// TIA Portal V20 export
DATA_BLOCK "ControlNodes"   // DB77
{ DB_Accessible_From_OPC_UA := 'FALSE' }
AUTHOR : ERsystem_FA2_DH. Kim
// stored: DBAccessibleFromOPCUA false, DBAccessibleFromWebserver false, MemoryReserve 100, Namespace Unit1.Em3
   VAR
      em { ExternalWritable := 'False'} : "LAF_typeEmControlNode";
      cm : Struct
         Interlock : Struct
            compensatorAxisX : "LER_typeAxisInterlock";
            masterVirtualAxis : "LER_typeAxisInterlock";
            unwinderVirtualAxis : "LER_typeAxisInterlock";
            dancerFwdBwd : "LER_typeTwoWayActInterlock";
            sepaUnwinderIonizerTop : "LER_typeTwoWayActInterlock";
            sepaUnwinderIonizerBottom : "LER_typeTwoWayActInterlock";
         END_STRUCT;
         command : Struct
            compensatorAxisX : "LER_typeAxisCommand";
            masterVirtualAxis : "LER_typeAxisCommand";
            unwinderVirtualAxis : "LER_typeAxisCommand";
            dancerFwdBwd : "LER_typeTwoWayActCommand";
            sepaUnwinderIonizerTop : "LER_typeTwoWayActCommand";
            sepaUnwinderIonizerBottom : "LER_typeTwoWayActCommand";
         END_STRUCT;
         softCam : "Unit1.type_emRelations_em3_SoftCam";
      END_STRUCT;
      citiMap : "LER_OEM_Data";
      webGuide : Struct
         jobs : "LAF_typeJobs";
         sequence : "LAF_typeSequence";
         "step" : "LER_typeStep";
         jobInterface : Struct
            null : Bool;
         END_STRUCT;
         preOperationCheck : Struct
            home : Bool;
            Bool2 : Bool;
            Bool3 : Bool;
            Bool4 : Bool;
            Bool5 : Bool;
            Bool6 : Bool;
            Bool7 : Bool;
            Bool8 : Bool;
            Bool9 : Bool;
            Bool10 : Bool;
            Bool11 : Bool;
            Bool12 : Bool;
            Bool13 : Bool;
            Bool14 : Bool;
            Bool15 : Bool;
            Bool16 : Bool;
            Bool17 : Bool;
            Bool18 : Bool;
            Bool19 : Bool;
            Bool20 : Bool;
         END_STRUCT;
      END_STRUCT;
      emRelations : Struct
         em2 : Struct
            reqDancerOn : Bool;
            reqDancerOff : Bool;
         END_STRUCT;
      END_STRUCT;
      cmSafetyPinIdlePositionSensor : "LBC_typeDigitalSignalControlNode";
      cmRotationSafetyPinPositionSensor : "LBC_typeDigitalSignalControlNode";
      cmIonizerTopMaintDetection : "LBC_typeDigitalSignalControlNode";
      cmIonizerTopErrorDetection : "LBC_typeDigitalSignalControlNode";
      cmIonizerBtmMaintDetection : "LBC_typeDigitalSignalControlNode";
      cmIonizerBtmErrorDetection : "LBC_typeDigitalSignalControlNode";
      cmDancerEncoder { ExternalAccessible := 'False'; ExternalVisible := 'False'; ExternalWritable := 'False'} : "LBC_typeAnalogInputControlNode";
      cmLoadCellControllerInterface { ExternalAccessible := 'False'; ExternalVisible := 'False'; ExternalWritable := 'False'} : "LBC_typeAnalogInputControlNode";
      cmDancerElectroPneumaticRegulator { ExternalAccessible := 'False'; ExternalVisible := 'False'; ExternalWritable := 'False'} : "LBC_typeAnalogOutputControlNode";
      cmCompensatorAxisX { ExternalAccessible := 'False'; ExternalVisible := 'False'; ExternalWritable := 'False'} : "LBC_typeAxis64PosControlNode";
      cmUnwinderVirtualAxis { ExternalAccessible := 'False'; ExternalVisible := 'False'; ExternalWritable := 'False'} : "LBC_typeAxis64PosControlNode";
      cmDancerFwdBwd { ExternalAccessible := 'False'; ExternalVisible := 'False'; ExternalWritable := 'False'} : "LBC_typeTwoWayActuatorControlNode";
      cmSepaUnwinderIonizerTop { ExternalAccessible := 'False'; ExternalVisible := 'False'; ExternalWritable := 'False'} : "LBC_typeTwoWayActuatorControlNode";
      cmSepaUnwinderIonizerBottom { ExternalAccessible := 'False'; ExternalVisible := 'False'; ExternalWritable := 'False'} : "LBC_typeTwoWayActuatorControlNode";
      cmEpcPivot { ExternalAccessible := 'False'; ExternalVisible := 'False'; ExternalWritable := 'False'} : "LER_typeCON600ControlNode";
   END_VAR
BEGIN
   em.commands.enable := FALSE;
   em.commands.acknowledge := FALSE;
   em.commands.disableAlarms := FALSE;
   em.commands.activateSimulation := FALSE;
   em.commands.home := FALSE;
   em.commands.moveToInitialPosition := FALSE;
   em.commands.directModeControl.current := 2;
   em.commands.directModeControl.production := FALSE;
   em.commands.directModeControl.maintenance := TRUE;
   em.commands.directModeControl.manual := FALSE;
   em.commands.directModeControl.nomode := FALSE;
   em.commands.directModeControl.sleep := FALSE;
   em.commands.directModeControl.deepsleep := FALSE;
   em.commands.directModeControl.userMode04 := FALSE;
   em.commands.directModeControl.userMode05 := FALSE;
   em.commands.directModeControl.userMode06 := FALSE;
   em.commands.directModeControl.userMode07 := FALSE;
   em.commands.directModeControl.userMode08 := FALSE;
   em.commands.directModeControl.userMode09 := FALSE;
   em.commands.directModeControl.userMode10 := FALSE;
   em.commands.directModeControl.userMode11 := FALSE;
   em.commands.directModeControl.userMode12 := FALSE;
   em.commands.directModeControl.userMode13 := FALSE;
   em.commands.directStateControl.current := 2;
   em.commands.directStateControl.clearing := FALSE;
   em.commands.directStateControl.stopped := TRUE;
   em.commands.directStateControl.starting := FALSE;
   em.commands.directStateControl.idle := FALSE;
   em.commands.directStateControl.suspended := FALSE;
   em.commands.directStateControl.execute := FALSE;
   em.commands.directStateControl.stopping := FALSE;
   em.commands.directStateControl.aborting := FALSE;
   em.commands.directStateControl.aborted := FALSE;
   em.commands.directStateControl.holding := FALSE;
   em.commands.directStateControl.held := FALSE;
   em.commands.directStateControl.unholding := FALSE;
   em.commands.directStateControl.suspending := FALSE;
   em.commands.directStateControl.unsuspending := FALSE;
   em.commands.directStateControl.resetting := FALSE;
   em.commands.directStateControl.completing := FALSE;
   em.commands.directStateControl.complete := FALSE;
   em.status.enabled := TRUE;
   em.status.acknowledgeActive := FALSE;
   em.status.alarmsDisabled := FALSE;
   em.status.simulationActive := FALSE;
   em.status.safetyReleased := TRUE;
   em.status.initialized := FALSE;
   em.status.homed := TRUE;
   em.status.safeState := FALSE;
   em.status.stateComplete := TRUE;
   // webGuide."step".action1[101] : Step[101] : JOB[1] Condition
   // webGuide."step".action1[110] : Step[110] : Ionizer On
   // webGuide."step".action1[120] : Step[120] : Web Guide EPC Mode Check
   // webGuide."step".action1[130] : Step[130] : Dancer On
   // webGuide."step".action1[180] : Step[180] : Compansator X-Axis WaitPos
   // webGuide."step".action1[190] : Step[190] : Job[1] Step End
   // webGuide."step".action1[201] : Step[201] : JOB[2] Condition
   // webGuide."step".action1[280] : Step[280] : Compansator X-Axis Compensation [Motion]
   // webGuide."step".action1[290] : Step[290] : Job[2] Step End
   // webGuide."step".transition1[101] : Step[101] : JOB[1] Condition
   // webGuide."step".transition1[110] : Step[110] : Ionizer On
   // webGuide."step".transition1[120] : Step[120] : Web Guide EPC Mode Check
   // webGuide."step".transition1[130] : Step[130] : Dancer On
   // webGuide."step".transition1[180] : Step[180] : Compansator X-Axis WaitPos
   // webGuide."step".transition1[190] : Step[190] : Job[1] Step End
   // webGuide."step".transition1[201] : Step[201] : JOB[2] Condition
   // webGuide."step".transition1[280] : Step[280] : Compansator X-Axis Compensation [Motion]
   // webGuide."step".transition1[290] : Step[290] : Job[2] Step End
   cmSafetyPinIdlePositionSensor.commands.reset := FALSE;
   cmSafetyPinIdlePositionSensor.commands.simulation := FALSE;
   cmSafetyPinIdlePositionSensor.commands.quality := TRUE;
   cmSafetyPinIdlePositionSensor.monitoring.valid := TRUE;
   cmSafetyPinIdlePositionSensor.monitoring.busy := TRUE;
   cmSafetyPinIdlePositionSensor.monitoring.error := FALSE;
   cmSafetyPinIdlePositionSensor.monitoring.status := 16#0000;
   cmSafetyPinIdlePositionSensor.monitoring.risingEdge := FALSE;
   cmSafetyPinIdlePositionSensor.monitoring.fallingEdge := FALSE;
   cmSafetyPinIdlePositionSensor.monitoring.processValue := TRUE;
   cmRotationSafetyPinPositionSensor.commands.reset := FALSE;
   cmRotationSafetyPinPositionSensor.commands.simulation := FALSE;
   cmRotationSafetyPinPositionSensor.commands.quality := TRUE;
   cmRotationSafetyPinPositionSensor.monitoring.valid := TRUE;
   cmRotationSafetyPinPositionSensor.monitoring.busy := TRUE;
   cmRotationSafetyPinPositionSensor.monitoring.error := FALSE;
   cmRotationSafetyPinPositionSensor.monitoring.status := 16#0000;
   cmRotationSafetyPinPositionSensor.monitoring.risingEdge := FALSE;
   cmRotationSafetyPinPositionSensor.monitoring.fallingEdge := FALSE;
   cmRotationSafetyPinPositionSensor.monitoring.processValue := TRUE;
   cmIonizerTopMaintDetection.commands.reset := FALSE;
   cmIonizerTopMaintDetection.commands.simulation := FALSE;
   cmIonizerTopMaintDetection.commands.quality := TRUE;
   cmIonizerTopMaintDetection.monitoring.valid := TRUE;
   cmIonizerTopMaintDetection.monitoring.busy := TRUE;
   cmIonizerTopMaintDetection.monitoring.error := FALSE;
   cmIonizerTopMaintDetection.monitoring.status := 16#0000;
   cmIonizerTopMaintDetection.monitoring.risingEdge := FALSE;
   cmIonizerTopMaintDetection.monitoring.fallingEdge := FALSE;
   cmIonizerTopMaintDetection.monitoring.processValue := FALSE;
   cmIonizerTopErrorDetection.commands.reset := FALSE;
   cmIonizerTopErrorDetection.commands.simulation := FALSE;
   cmIonizerTopErrorDetection.commands.quality := TRUE;
   cmIonizerTopErrorDetection.monitoring.valid := TRUE;
   cmIonizerTopErrorDetection.monitoring.busy := TRUE;
   cmIonizerTopErrorDetection.monitoring.error := FALSE;
   cmIonizerTopErrorDetection.monitoring.status := 16#0000;
   cmIonizerTopErrorDetection.monitoring.risingEdge := FALSE;
   cmIonizerTopErrorDetection.monitoring.fallingEdge := FALSE;
   cmIonizerTopErrorDetection.monitoring.processValue := TRUE;
   cmIonizerBtmMaintDetection.commands.reset := FALSE;
   cmIonizerBtmMaintDetection.commands.simulation := FALSE;
   cmIonizerBtmMaintDetection.commands.quality := TRUE;
   cmIonizerBtmMaintDetection.monitoring.valid := TRUE;
   cmIonizerBtmMaintDetection.monitoring.busy := TRUE;
   cmIonizerBtmMaintDetection.monitoring.error := FALSE;
   cmIonizerBtmMaintDetection.monitoring.status := 16#0000;
   cmIonizerBtmMaintDetection.monitoring.risingEdge := FALSE;
   cmIonizerBtmMaintDetection.monitoring.fallingEdge := FALSE;
   cmIonizerBtmMaintDetection.monitoring.processValue := FALSE;
   cmIonizerBtmErrorDetection.commands.reset := FALSE;
   cmIonizerBtmErrorDetection.commands.simulation := FALSE;
   cmIonizerBtmErrorDetection.commands.quality := TRUE;
   cmIonizerBtmErrorDetection.monitoring.valid := TRUE;
   cmIonizerBtmErrorDetection.monitoring.busy := TRUE;
   cmIonizerBtmErrorDetection.monitoring.error := FALSE;
   cmIonizerBtmErrorDetection.monitoring.status := 16#0000;
   cmIonizerBtmErrorDetection.monitoring.risingEdge := FALSE;
   cmIonizerBtmErrorDetection.monitoring.fallingEdge := FALSE;
   cmIonizerBtmErrorDetection.monitoring.processValue := TRUE;
   cmCompensatorAxisX.commandConfiguration.power.startMode := 1;
   cmCompensatorAxisX.commandConfiguration.power.stopMode := 0;
   cmCompensatorAxisX.commandConfiguration.power.syncMotionSimulation := FALSE;
   cmCompensatorAxisX.commandConfiguration.power.syncMotionSimulationExtendedMode := -1;
   cmCompensatorAxisX.commandConfiguration.jog.velocity := 0.0;
   cmCompensatorAxisX.commandConfiguration.jog.acceleration := -1.0;
   cmCompensatorAxisX.commandConfiguration.jog.deceleration := -1.0;
   cmCompensatorAxisX.commandConfiguration.jog.jerk := -1.0;
   cmCompensatorAxisX.commandConfiguration.jog.positionControlled := TRUE;
   cmCompensatorAxisX.commandConfiguration.jog.increment := 0.0;
   cmCompensatorAxisX.commandConfiguration.jog.mode := 0;
   cmCompensatorAxisX.commandConfiguration.moveVelocity.velocity := 0.0;
   cmCompensatorAxisX.commandConfiguration.moveVelocity.acceleration := -1.0;
   cmCompensatorAxisX.commandConfiguration.moveVelocity.deceleration := -1.0;
   cmCompensatorAxisX.commandConfiguration.moveVelocity.jerk := -1.0;
   cmCompensatorAxisX.commandConfiguration.moveVelocity.direction := 0;
   cmCompensatorAxisX.commandConfiguration.moveVelocity.positionControlled := TRUE;
   cmCompensatorAxisX.commandConfiguration.moveVelocity.velocityChangeOnTheFly := FALSE;
   cmCompensatorAxisX.commandConfiguration.stop.deceleration := -1.0;
   cmCompensatorAxisX.commandConfiguration.stop.jerk := -1.0;
   cmCompensatorAxisX.commandConfiguration.stop.abortAcceleration := FALSE;
   cmCompensatorAxisX.commandConfiguration.fastStop.deceleration := -1.0;
   cmCompensatorAxisX.commandConfiguration.fastStop.jerk := -1.0;
   cmCompensatorAxisX.commandConfiguration.fastStop.abortAcceleration := FALSE;
   cmCompensatorAxisX.commandConfiguration.fastStop.replaceStopPossible := FALSE;
   cmCompensatorAxisX.commandConfiguration.torqueLimiting.limit := -1.0;
   cmCompensatorAxisX.commandConfiguration.torqueLimiting.mode := 0;
   cmCompensatorAxisX.commandConfiguration.homing.position := 0.0;
   cmCompensatorAxisX.commandConfiguration.homing.mode := 0;
   cmCompensatorAxisX.commandConfiguration.homing.sensor := 0;
   cmCompensatorAxisX.commandConfiguration.homing.extendedMode := -1;
   cmCompensatorAxisX.commandConfiguration.homing.extendedModeTorqueLimit := 0.0;
   cmCompensatorAxisX.commandConfiguration.homing.extendedModeTargetPosition := 0.0;
   cmCompensatorAxisX.commandConfiguration.posRelative.distance := 0.0;
   cmCompensatorAxisX.commandConfiguration.posRelative.velocity := -1.0;
   cmCompensatorAxisX.commandConfiguration.posRelative.acceleration := -1.0;
   cmCompensatorAxisX.commandConfiguration.posRelative.deceleration := -1.0;
   cmCompensatorAxisX.commandConfiguration.posRelative.jerk := -1.0;
   cmCompensatorAxisX.commandConfiguration.posRelative.direction := 0;
   cmCompensatorAxisX.commandConfiguration.posAbsolute.position := 0.0;
   cmCompensatorAxisX.commandConfiguration.posAbsolute.velocity := -1.0;
   cmCompensatorAxisX.commandConfiguration.posAbsolute.acceleration := -1.0;
   cmCompensatorAxisX.commandConfiguration.posAbsolute.deceleration := -1.0;
   cmCompensatorAxisX.commandConfiguration.posAbsolute.jerk := -1.0;
   cmCompensatorAxisX.commandConfiguration.posAbsolute.direction := 1;
   cmCompensatorAxisX.commandConfiguration.posAbsolute.positionChangeOnTheFly := FALSE;
   cmCompensatorAxisX.commandConfiguration.posAbsolute.velocityChangeOnTheFly := FALSE;
   cmCompensatorAxisX.commandConfiguration.posSuperimposed.distance := 0.0;
   cmCompensatorAxisX.commandConfiguration.posSuperimposed.velocityDiff := -1.0;
   cmCompensatorAxisX.commandConfiguration.posSuperimposed.acceleration := -1.0;
   cmCompensatorAxisX.commandConfiguration.posSuperimposed.deceleration := -1.0;
   cmCompensatorAxisX.commandConfiguration.posSuperimposed.jerk := -1.0;
   cmCompensatorAxisX.commandConfiguration.posSuperimposed.direction := 0;
   cmCompensatorAxisX.commandConfiguration.haltSuperimposed.deceleration := -1.0;
   cmCompensatorAxisX.commandConfiguration.haltSuperimposed.jerk := -1.0;
   cmCompensatorAxisX.commandConfiguration.haltSuperimposed.abortAcceleration := FALSE;
   cmCompensatorAxisX.commandConfiguration.gearInRelative.ratioNumerator := 1;
   cmCompensatorAxisX.commandConfiguration.gearInRelative.ratioDenominator := 1;
   cmCompensatorAxisX.commandConfiguration.gearInRelative.acceleration := -1.0;
   cmCompensatorAxisX.commandConfiguration.gearInRelative.deceleration := -1.0;
   cmCompensatorAxisX.commandConfiguration.gearInRelative.jerk := -1.0;
   cmCompensatorAxisX.commandConfiguration.gearInRelative.ratioChangeOnTheFly := FALSE;
   cmCompensatorAxisX.commandConfiguration.gearInAbsolute.ratioNumerator := 1;
   cmCompensatorAxisX.commandConfiguration.gearInAbsolute.ratioDenominator := 1;
   cmCompensatorAxisX.commandConfiguration.gearInAbsolute.masterSyncPosition := 0.0;
   cmCompensatorAxisX.commandConfiguration.gearInAbsolute.slaveSyncPosition := 0.0;
   cmCompensatorAxisX.commandConfiguration.gearInAbsolute.syncProfileReference := 1;
   cmCompensatorAxisX.commandConfiguration.gearInAbsolute.masterStartDistance := 0.0;
   cmCompensatorAxisX.commandConfiguration.gearInAbsolute.velocity := -1.0;
   cmCompensatorAxisX.commandConfiguration.gearInAbsolute.acceleration := -1.0;
   cmCompensatorAxisX.commandConfiguration.gearInAbsolute.deceleration := -1.0;
   cmCompensatorAxisX.commandConfiguration.gearInAbsolute.jerk := -1.0;
   cmCompensatorAxisX.commandConfiguration.gearInAbsolute.syncDirection := 1;
   cmCompensatorAxisX.commandConfiguration.gearInAbsolute.ratioChangeOnTheFly := FALSE;
   cmCompensatorAxisX.commandConfiguration.gearInVelocity.continuousUpdate := FALSE;
   cmCompensatorAxisX.commandConfiguration.gearInVelocity.ratioNumerator := 1;
   cmCompensatorAxisX.commandConfiguration.gearInVelocity.ratioDenominator := 1;
   cmCompensatorAxisX.commandConfiguration.gearInVelocity.acceleration := -1.0;
   cmCompensatorAxisX.commandConfiguration.gearInVelocity.deceleration := -1.0;
   cmCompensatorAxisX.commandConfiguration.gearInVelocity.jerk := -1.0;
   cmCompensatorAxisX.commandConfiguration.gearInVelocity.positionControlled := FALSE;
   cmCompensatorAxisX.commandConfiguration.camIn.masterOffset := 0.0;
   cmCompensatorAxisX.commandConfiguration.camIn.slaveOffset := 0.0;
   cmCompensatorAxisX.commandConfiguration.camIn.masterScaling := 1.0;
   cmCompensatorAxisX.commandConfiguration.camIn.slaveScaling := 1.0;
   cmCompensatorAxisX.commandConfiguration.camIn.masterSyncPosition := 0.0;
   cmCompensatorAxisX.commandConfiguration.camIn.syncProfileReference := 1;
   cmCompensatorAxisX.commandConfiguration.camIn.masterStartDistance := 0.0;
   cmCompensatorAxisX.commandConfiguration.camIn.velocity := -1.0;
   cmCompensatorAxisX.commandConfiguration.camIn.acceleration := -1.0;
   cmCompensatorAxisX.commandConfiguration.camIn.deceleration := -1.0;
   cmCompensatorAxisX.commandConfiguration.camIn.jerk := -1.0;
   cmCompensatorAxisX.commandConfiguration.camIn.applicationMode := 0;
   cmCompensatorAxisX.commandConfiguration.camIn.syncDirection := 1;
   cmCompensatorAxisX.commandConfiguration.gearOutCamOut.slavePosition := 0.0;
   cmCompensatorAxisX.commandConfiguration.gearOutCamOut.syncProfileReference := 1;
   cmCompensatorAxisX.commandConfiguration.gearOutCamOut.masterStopDistance := 0.0;
   cmCompensatorAxisX.commandConfiguration.gearOutCamOut.deceleration := -1.0;
   cmCompensatorAxisX.commandConfiguration.gearOutCamOut.jerk := -1.0;
   cmCompensatorAxisX.commandConfiguration.gearOutCamOut.syncOutDirection := 3;
   cmCompensatorAxisX.commandConfiguration.gearOutCamOut.gearOutCamOutMode := -1;
   cmCompensatorAxisX.commandConfiguration.phasing.phaseShift := 0.0;
   cmCompensatorAxisX.commandConfiguration.phasing.velocity := -1.0;
   cmCompensatorAxisX.commandConfiguration.phasing.acceleration := -1.0;
   cmCompensatorAxisX.commandConfiguration.phasing.deceleration := -1.0;
   cmCompensatorAxisX.commandConfiguration.phasing.jerk := -1.0;
   cmCompensatorAxisX.commandConfiguration.phasing.profileReference := 0;
   cmCompensatorAxisX.commandConfiguration.phasing.phasingDistance := 0.0;
   cmCompensatorAxisX.commandConfiguration.phasing.startPosition := 0.0;
   cmCompensatorAxisX.commandConfiguration.phasing.direction := 3;
   cmCompensatorAxisX.commandConfiguration.phasing.phaseAbsolute := TRUE;
   cmCompensatorAxisX.commandConfiguration.phasing.phaseShiftChangeOnTheFly := FALSE;
   cmCompensatorAxisX.commandConfiguration.offset.offset := 0.0;
   cmCompensatorAxisX.commandConfiguration.offset.profileReference := 1;
   cmCompensatorAxisX.commandConfiguration.offset.offsetDistance := 0.0;
   cmCompensatorAxisX.commandConfiguration.offset.startPosition := 0.0;
   cmCompensatorAxisX.commandConfiguration.offset.direction := 3;
   cmCompensatorAxisX.commandConfiguration.offset.offsetAbsolute := TRUE;
   cmCompensatorAxisX.commandConfiguration.offset.offsetChangeOnTheFly := FALSE;
   cmUnwinderVirtualAxis.commandConfiguration.power.startMode := 1;
   cmUnwinderVirtualAxis.commandConfiguration.power.stopMode := 0;
   cmUnwinderVirtualAxis.commandConfiguration.power.syncMotionSimulation := FALSE;
   cmUnwinderVirtualAxis.commandConfiguration.power.syncMotionSimulationExtendedMode := -1;
   cmUnwinderVirtualAxis.commandConfiguration.jog.velocity := 0.0;
   cmUnwinderVirtualAxis.commandConfiguration.jog.acceleration := -1.0;
   cmUnwinderVirtualAxis.commandConfiguration.jog.deceleration := -1.0;
   cmUnwinderVirtualAxis.commandConfiguration.jog.jerk := -1.0;
   cmUnwinderVirtualAxis.commandConfiguration.jog.positionControlled := TRUE;
   cmUnwinderVirtualAxis.commandConfiguration.jog.increment := 0.0;
   cmUnwinderVirtualAxis.commandConfiguration.jog.mode := 0;
   cmUnwinderVirtualAxis.commandConfiguration.moveVelocity.velocity := 0.0;
   cmUnwinderVirtualAxis.commandConfiguration.moveVelocity.acceleration := -1.0;
   cmUnwinderVirtualAxis.commandConfiguration.moveVelocity.deceleration := -1.0;
   cmUnwinderVirtualAxis.commandConfiguration.moveVelocity.jerk := -1.0;
   cmUnwinderVirtualAxis.commandConfiguration.moveVelocity.direction := 0;
   cmUnwinderVirtualAxis.commandConfiguration.moveVelocity.positionControlled := TRUE;
   cmUnwinderVirtualAxis.commandConfiguration.moveVelocity.velocityChangeOnTheFly := FALSE;
   cmUnwinderVirtualAxis.commandConfiguration.stop.deceleration := -1.0;
   cmUnwinderVirtualAxis.commandConfiguration.stop.jerk := -1.0;
   cmUnwinderVirtualAxis.commandConfiguration.stop.abortAcceleration := FALSE;
   cmUnwinderVirtualAxis.commandConfiguration.fastStop.deceleration := -1.0;
   cmUnwinderVirtualAxis.commandConfiguration.fastStop.jerk := -1.0;
   cmUnwinderVirtualAxis.commandConfiguration.fastStop.abortAcceleration := FALSE;
   cmUnwinderVirtualAxis.commandConfiguration.fastStop.replaceStopPossible := FALSE;
   cmUnwinderVirtualAxis.commandConfiguration.torqueLimiting.limit := -1.0;
   cmUnwinderVirtualAxis.commandConfiguration.torqueLimiting.mode := 0;
   cmUnwinderVirtualAxis.commandConfiguration.homing.position := 0.0;
   cmUnwinderVirtualAxis.commandConfiguration.homing.mode := 0;
   cmUnwinderVirtualAxis.commandConfiguration.homing.sensor := 0;
   cmUnwinderVirtualAxis.commandConfiguration.homing.extendedMode := -1;
   cmUnwinderVirtualAxis.commandConfiguration.homing.extendedModeTorqueLimit := 0.0;
   cmUnwinderVirtualAxis.commandConfiguration.homing.extendedModeTargetPosition := 0.0;
   cmUnwinderVirtualAxis.commandConfiguration.posRelative.distance := 0.0;
   cmUnwinderVirtualAxis.commandConfiguration.posRelative.velocity := -1.0;
   cmUnwinderVirtualAxis.commandConfiguration.posRelative.acceleration := -1.0;
   cmUnwinderVirtualAxis.commandConfiguration.posRelative.deceleration := -1.0;
   cmUnwinderVirtualAxis.commandConfiguration.posRelative.jerk := -1.0;
   cmUnwinderVirtualAxis.commandConfiguration.posRelative.direction := 0;
   cmUnwinderVirtualAxis.commandConfiguration.posAbsolute.position := 0.0;
   cmUnwinderVirtualAxis.commandConfiguration.posAbsolute.velocity := -1.0;
   cmUnwinderVirtualAxis.commandConfiguration.posAbsolute.acceleration := -1.0;
   cmUnwinderVirtualAxis.commandConfiguration.posAbsolute.deceleration := -1.0;
   cmUnwinderVirtualAxis.commandConfiguration.posAbsolute.jerk := -1.0;
   cmUnwinderVirtualAxis.commandConfiguration.posAbsolute.direction := 1;
   cmUnwinderVirtualAxis.commandConfiguration.posAbsolute.positionChangeOnTheFly := FALSE;
   cmUnwinderVirtualAxis.commandConfiguration.posAbsolute.velocityChangeOnTheFly := FALSE;
   cmUnwinderVirtualAxis.commandConfiguration.posSuperimposed.distance := 0.0;
   cmUnwinderVirtualAxis.commandConfiguration.posSuperimposed.velocityDiff := -1.0;
   cmUnwinderVirtualAxis.commandConfiguration.posSuperimposed.acceleration := -1.0;
   cmUnwinderVirtualAxis.commandConfiguration.posSuperimposed.deceleration := -1.0;
   cmUnwinderVirtualAxis.commandConfiguration.posSuperimposed.jerk := -1.0;
   cmUnwinderVirtualAxis.commandConfiguration.posSuperimposed.direction := 0;
   cmUnwinderVirtualAxis.commandConfiguration.haltSuperimposed.deceleration := -1.0;
   cmUnwinderVirtualAxis.commandConfiguration.haltSuperimposed.jerk := -1.0;
   cmUnwinderVirtualAxis.commandConfiguration.haltSuperimposed.abortAcceleration := FALSE;
   cmUnwinderVirtualAxis.commandConfiguration.gearInRelative.ratioNumerator := 1;
   cmUnwinderVirtualAxis.commandConfiguration.gearInRelative.ratioDenominator := 1;
   cmUnwinderVirtualAxis.commandConfiguration.gearInRelative.acceleration := -1.0;
   cmUnwinderVirtualAxis.commandConfiguration.gearInRelative.deceleration := -1.0;
   cmUnwinderVirtualAxis.commandConfiguration.gearInRelative.jerk := -1.0;
   cmUnwinderVirtualAxis.commandConfiguration.gearInRelative.ratioChangeOnTheFly := FALSE;
   cmUnwinderVirtualAxis.commandConfiguration.gearInAbsolute.ratioNumerator := 1;
   cmUnwinderVirtualAxis.commandConfiguration.gearInAbsolute.ratioDenominator := 1;
   cmUnwinderVirtualAxis.commandConfiguration.gearInAbsolute.masterSyncPosition := 0.0;
   cmUnwinderVirtualAxis.commandConfiguration.gearInAbsolute.slaveSyncPosition := 0.0;
   cmUnwinderVirtualAxis.commandConfiguration.gearInAbsolute.syncProfileReference := 1;
   cmUnwinderVirtualAxis.commandConfiguration.gearInAbsolute.masterStartDistance := 0.0;
   cmUnwinderVirtualAxis.commandConfiguration.gearInAbsolute.velocity := -1.0;
   cmUnwinderVirtualAxis.commandConfiguration.gearInAbsolute.acceleration := -1.0;
   cmUnwinderVirtualAxis.commandConfiguration.gearInAbsolute.deceleration := -1.0;
   cmUnwinderVirtualAxis.commandConfiguration.gearInAbsolute.jerk := -1.0;
   cmUnwinderVirtualAxis.commandConfiguration.gearInAbsolute.syncDirection := 1;
   cmUnwinderVirtualAxis.commandConfiguration.gearInAbsolute.ratioChangeOnTheFly := FALSE;
   cmUnwinderVirtualAxis.commandConfiguration.gearInVelocity.continuousUpdate := FALSE;
   cmUnwinderVirtualAxis.commandConfiguration.gearInVelocity.ratioNumerator := 1;
   cmUnwinderVirtualAxis.commandConfiguration.gearInVelocity.ratioDenominator := 1;
   cmUnwinderVirtualAxis.commandConfiguration.gearInVelocity.acceleration := -1.0;
   cmUnwinderVirtualAxis.commandConfiguration.gearInVelocity.deceleration := -1.0;
   cmUnwinderVirtualAxis.commandConfiguration.gearInVelocity.jerk := -1.0;
   cmUnwinderVirtualAxis.commandConfiguration.gearInVelocity.positionControlled := FALSE;
   cmUnwinderVirtualAxis.commandConfiguration.camIn.masterOffset := 0.0;
   cmUnwinderVirtualAxis.commandConfiguration.camIn.slaveOffset := 0.0;
   cmUnwinderVirtualAxis.commandConfiguration.camIn.masterScaling := 1.0;
   cmUnwinderVirtualAxis.commandConfiguration.camIn.slaveScaling := 1.0;
   cmUnwinderVirtualAxis.commandConfiguration.camIn.masterSyncPosition := 0.0;
   cmUnwinderVirtualAxis.commandConfiguration.camIn.syncProfileReference := 1;
   cmUnwinderVirtualAxis.commandConfiguration.camIn.masterStartDistance := 0.0;
   cmUnwinderVirtualAxis.commandConfiguration.camIn.velocity := -1.0;
   cmUnwinderVirtualAxis.commandConfiguration.camIn.acceleration := -1.0;
   cmUnwinderVirtualAxis.commandConfiguration.camIn.deceleration := -1.0;
   cmUnwinderVirtualAxis.commandConfiguration.camIn.jerk := -1.0;
   cmUnwinderVirtualAxis.commandConfiguration.camIn.applicationMode := 0;
   cmUnwinderVirtualAxis.commandConfiguration.camIn.syncDirection := 1;
   cmUnwinderVirtualAxis.commandConfiguration.gearOutCamOut.slavePosition := 0.0;
   cmUnwinderVirtualAxis.commandConfiguration.gearOutCamOut.syncProfileReference := 1;
   cmUnwinderVirtualAxis.commandConfiguration.gearOutCamOut.masterStopDistance := 0.0;
   cmUnwinderVirtualAxis.commandConfiguration.gearOutCamOut.deceleration := -1.0;
   cmUnwinderVirtualAxis.commandConfiguration.gearOutCamOut.jerk := -1.0;
   cmUnwinderVirtualAxis.commandConfiguration.gearOutCamOut.syncOutDirection := 3;
   cmUnwinderVirtualAxis.commandConfiguration.gearOutCamOut.gearOutCamOutMode := -1;
   cmUnwinderVirtualAxis.commandConfiguration.phasing.phaseShift := 0.0;
   cmUnwinderVirtualAxis.commandConfiguration.phasing.velocity := -1.0;
   cmUnwinderVirtualAxis.commandConfiguration.phasing.acceleration := -1.0;
   cmUnwinderVirtualAxis.commandConfiguration.phasing.deceleration := -1.0;
   cmUnwinderVirtualAxis.commandConfiguration.phasing.jerk := -1.0;
   cmUnwinderVirtualAxis.commandConfiguration.phasing.profileReference := 0;
   cmUnwinderVirtualAxis.commandConfiguration.phasing.phasingDistance := 0.0;
   cmUnwinderVirtualAxis.commandConfiguration.phasing.startPosition := 0.0;
   cmUnwinderVirtualAxis.commandConfiguration.phasing.direction := 3;
   cmUnwinderVirtualAxis.commandConfiguration.phasing.phaseAbsolute := TRUE;
   cmUnwinderVirtualAxis.commandConfiguration.phasing.phaseShiftChangeOnTheFly := FALSE;
   cmUnwinderVirtualAxis.commandConfiguration.offset.offset := 0.0;
   cmUnwinderVirtualAxis.commandConfiguration.offset.profileReference := 1;
   cmUnwinderVirtualAxis.commandConfiguration.offset.offsetDistance := 0.0;
   cmUnwinderVirtualAxis.commandConfiguration.offset.startPosition := 0.0;
   cmUnwinderVirtualAxis.commandConfiguration.offset.direction := 3;
   cmUnwinderVirtualAxis.commandConfiguration.offset.offsetAbsolute := TRUE;
   cmUnwinderVirtualAxis.commandConfiguration.offset.offsetChangeOnTheFly := FALSE;
END_DATA_BLOCK
